SUBAPPLICATION A2X_TO_A2X_AX (* Wie AX_2_TO_3, aber gebuendelt: A2X (UP/DOWN) durchgereicht + gemeinsames ODER (z.B. Treiber-Enable) als zusaetzliches AX-Signal *)
  (* Standard: 61499-2; Description: Copyright (c) 2026 Meisterschulen am Ostbahnhof This program and the accompanying materials are made available under the terms of the Eclipse Public License 2.0 which is available at https://www.eclipse.org/legal/epl-2.0/ SPDX-License-Identifier: EPL-2.0 *)
  (* Version 1.0, 2026-09-06, Franz Höpfinger, Meisterschulen am Ostbahnhof, initial API and implementation and/or initial documentation *)
  PACKAGE MyLib::sys;
  (* Documentation:
  A2X-Passthrough plus gemeinsames ODER als zusätzliches AX-Signal
   Gebündeltes Pendant zu AX_2_TO_3: statt zwei getrennter AX-Sockets/Plugs (UP_IN/DOWN_IN, UP_OUT/DOWN_OUT) nimmt dieser Baustein UP/DOWN gebündelt als ein einziges A2X-Signal entgegen und gibt sie ebenso gebündelt wieder aus - plus ein zusätzliches, einzelnes AX-Signal mit dem ODER aus beiden Richtungen.
   Funktionsbeschreibung
    - UNBUNDLE (A2X_2X_TO_2AX) trennt das eingehende A2X_IN in zwei einzelne AX-Signale (UP, DOWN) auf.
   - Je ein AX_SPLIT_2 pro Richtung, weil jedes der beiden Signale zu zwei Zielen muss: zurück ins gebündelte Ausgangssignal UND in die ODER-Verknüpfung.
   - BUNDLE (A2X_2AX_TO_2X) fügt UP/DOWN wieder zu einem einzigen A2X_OUT zusammen - nach außen bleibt die Bündelung erhalten, intern wird trotzdem unverändert durchgereicht wie bei AX_2_TO_3.
   - AX_OR_2 liefert auf OR_OUT "läuft der Aktor gerade in irgendeine Richtung" - z.B. für einen gemeinsamen Treiber/Enable-Ausgang.
    Verwenden, wenn UP/DOWN im Rest der Schaltung ohnehin als gebündeltes A2X geführt werden (z.B. Richtung an einem Doppelwirkungs-Ventil) und nicht extra in zwei einzelne AX-Signale aufgesplittet werden sollen. Werden UP/DOWN ohnehin einzeln als AX geführt, AX_2_TO_3 verwenden.
  *)
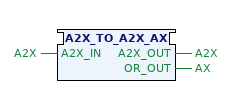
  SOCKETS
    A2X_IN : adapter::types::unidirectional::A2X; (* Gebuendeltes UP/DOWN Eingangssignal *)
  END_SOCKETS
  PLUGS
    A2X_OUT : adapter::types::unidirectional::A2X; (* Gebuendeltes UP/DOWN Ausgangssignal (unveraendert durchgereicht) *)
    OR_OUT : adapter::types::unidirectional::AX; (* ODER aus UP und DOWN *)
  END_PLUGS
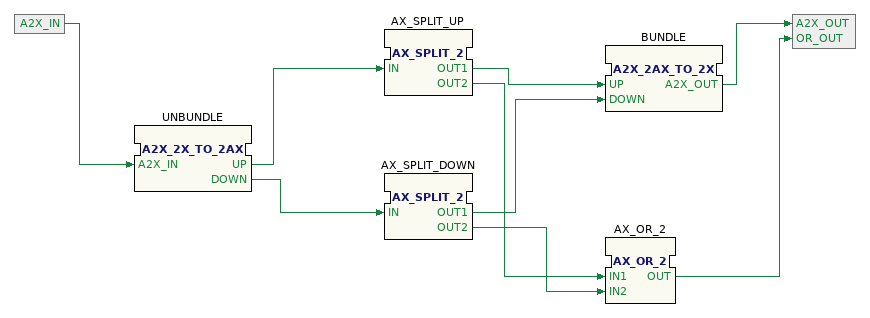
  FBS
    UNBUNDLE : adapter::conversion::unidirectional::A2X_2X_TO_2AX;
    AX_SPLIT_UP : adapter::events::unidirectional::AX_SPLIT_2;
    AX_SPLIT_DOWN : adapter::events::unidirectional::AX_SPLIT_2;
    BUNDLE : adapter::conversion::unidirectional::A2X_2AX_TO_2X;
    AX_OR_2 : adapter::booleanOperators::AX_OR_2;
  END_FBS
  ADAPTER_CONNECTIONS
    A2X_IN TO UNBUNDLE.A2X_IN;
    UNBUNDLE.UP TO AX_SPLIT_UP.IN;
    UNBUNDLE.DOWN TO AX_SPLIT_DOWN.IN;
    AX_SPLIT_UP.OUT1 TO BUNDLE.UP;
    AX_SPLIT_DOWN.OUT1 TO BUNDLE.DOWN;
    AX_SPLIT_UP.OUT2 TO AX_OR_2.IN1;
    AX_SPLIT_DOWN.OUT2 TO AX_OR_2.IN2;
    BUNDLE.A2X_OUT TO A2X_OUT;
    AX_OR_2.OUT TO OR_OUT;
  END_CONNECTIONS
END_SUBAPPLICATION
